KUKA KRL program: InitVariables.src

&ACCESS RVO
&REL 1167
&PARAM DISKPATH = KRC:\R1\Program\KUKA\Subprogs
DEF InitVariables ( )

   gbToolAlowedToUse[1]=TRUE
   gbToolAlowedToUse[2]=TRUE
   gbToolAlowedToUse[3]=TRUE

END
